TYPE
  (* Version 1.0, 2023-03-15, Tim Hesse *)
  ROS2_action_msgs__msg__GoalInfo : STRUCT
    goal_id : ROS2_unique_identifiers__msg__UUID;
    stamp : ROS2_builtin_interfaces__msg__Time;
  END_STRUCT;
END_TYPE
